FUNCTION F_VerifySBGaugeReadings : BOOL
VAR_INPUT
	stExpReadings : ST_SBGaugeReadings;
	stReadingsOp : ST_SBGaugeReadingsOp;
END_VAR
VAR
	stStatus : ST_SBGaugeReadings;
END_VAR

stStatus := F_GetSBGaugeReadings();

// Return true if the expected status matches the actual status
F_VerifySBGaugeReadings := 
	F_CompareGauge(
		eCompOp := stReadingsOp.eDPColdCathodeOp,
		fReading := stStatus.fDPColdCathodeVal,
		eState := stStatus.eDPColdCathodeState,
		fExpReading := stExpReadings.fDPColdCathodeVal,
		eExpState := stExpReadings.eDPColdCathodeState) 
	AND F_CompareGauge(
		eCompOp := stReadingsOp.eDPPiraniOp,
		fReading := stStatus.fDPPiraniVal,
		eState := stStatus.eDPPiraniState,
		fExpReading := stExpReadings.fDPPiraniVal,
		eExpState := stExpReadings.eDPPiraniState)
	AND F_CompareGauge(
		eCompOp := stReadingsOp.ePumpStationColdCathodeOp,
		fReading := stStatus.fPumpStationColdCathodeVal,
		eState := stStatus.ePumpStationColdCathodeState,
		fExpReading := stExpReadings.fPumpStationColdCathodeVal,
		eExpState := stExpReadings.ePumpStationColdCathodeState)
	AND F_CompareGauge(
		eCompOp := stReadingsOp.ePumpStationPirani1Op,
		fReading := stStatus.fPumpStationPirani1Val,
		eState := stStatus.ePumpStationPirani1State,
		fExpReading := stExpReadings.fPumpStationPirani1Val,
		eExpState := stExpReadings.ePumpStationPirani1State)
	AND F_CompareGauge(
		eCompOp := stReadingsOp.ePumpStationPirani2Op,
		fReading := stStatus.fPumpStationPirani2Val,
		eState := stStatus.ePumpStationPirani2State,
		fExpReading := stExpReadings.fPumpStationPirani2Val,
		eExpState := stExpReadings.ePumpStationPirani2State);

END_FUNCTION

(* stored: Version 1.1.0.1, ProductVersion 3.1.4024.0
   POU F_VerifySBGaugeReadings: Id {a066cf66-9a1e-46cb-b56b-9c11a5162294}, SpecialFunc None *)
